(* PLC project conveyor_v1.project, CODESYS CODESYS V3.5 SP22 Patch 3 *)
(* stored: creationDateTime 2026-09-17T14:55:14.2317014, modificationDateTime 2026-09-17T14:51:48.7175218 *)

PROGRAM PLC_PRG
  VAR
    bStart AT %IX0.0 : BOOL;  (* Nút Start (NO) *)
    bStop AT %IX0.1 : BOOL;  (* Nút Stop (NC) *)
    bSensor AT %IX0.2 : BOOL;  (* Cảm biến sản phẩm *)
    bReset AT %IX0.3 : BOOL;  (* Nút reset bộ đếm *)
    bMotor AT %QX0.0 : BOOL;  (* Contactor băng tải *)
    bLampRun AT %QX0.1 : BOOL;  (* Đèn báo chạy *)
    bLampDone AT %QX0.2 : BOOL;  (* Đèn báo đủ số lượng *)
  END_VAR
  VAR
    fbCounter : CTU;  (* Internal *)
    iCount : INT;
    iPreset : INT := 10;
  END_VAR

                    fbCounter(CU := bSensor AND bMotor, RESET := bReset, PV := iPreset,
          Q => bLampDone, CV => iCount);

bMotor   := (bStart OR bMotor) AND bStop AND NOT bLampDone;
bLampRun := bMotor;
                  
END_PROGRAM

CONFIGURATION Device
  RESOURCE Application ON PLC
    TASK MainTask(INTERVAL := T#20ms, PRIORITY := 1);
    PROGRAM PLC_PRG WITH MainTask : PLC_PRG;
  END_RESOURCE
END_CONFIGURATION
